Yaskawa INFORM job: R1_W39(90,0)R2.JBI

/JOB
//NAME R1_W39(90,0)R2
///FOLDERNAME KRIS-SCIANA
//POS
///NPOS 43,43,0,0,0,0
///TOOL 0
///POSTYPE PULSE
///PULSE
C00000=48919,5665,-78085,33957,84829,-60043
C00001=76192,72700,-3611,7580,89499,-58244
C00002=85002,90670,26729,6577,108191,-2594
C00003=82773,103392,47657,9044,108090,-2765
C00004=80348,95814,37890,14264,107528,-2580
C00005=80254,94172,37553,14217,106925,-2684
C00006=81389,106350,52541,15889,109549,-1922
C00007=88376,91776,33541,16145,112345,900
C00008=84647,97242,43547,26530,112715,1712
C00009=80535,96727,39662,19290,111179,-13264
C00010=80533,98698,38722,19533,112685,-13001
C00011=95804,88670,27983,-9101,104845,39456
C00012=93260,116784,65555,-9230,104296,50461
C00013=88788,88191,28703,620,100303,50675
C00014=93687,111856,59478,-9313,105536,50507
C00015=89184,93395,34979,471,102669,51670
C00016=95648,113896,64634,-12639,107588,50809
C00017=91118,114335,62249,-3400,106342,50920
C00018=94799,78029,20878,-7231,106457,51217
C00019=94179,105834,52955,-9270,106688,50794
C00020=97616,95145,42128,-15247,107009,50700
C00021=97568,79271,23775,-13354,106025,50913
C00022=97503,98351,37938,-14194,113675,56454
C00023=97503,100031,37397,-14345,114836,56304
C00024=130465,98764,47484,-38638,104472,-12047
C00025=128682,99899,51858,-38063,102058,-11895
C00026=125592,100494,53893,-37558,100021,-12435
C00027=117769,53841,-3568,-7004,89352,-33862
C00028=118319,55966,-2495,-7211,89822,-33727
C00029=127393,85542,37674,-37833,96354,-10529
C00030=118983,88052,33036,-15664,100505,-10201
C00031=114637,82539,25445,-1803,99860,-9026
C00032=114316,82458,25346,-216,99794,-11375
C00033=114685,80246,17709,-453,103292,-11364
C00034=111320,72755,14674,9080,100113,-13386
C00035=111645,74192,16353,7527,99507,-12765
C00036=112489,77538,20103,4175,98402,-12017
C00037=114786,72045,10431,-220,101192,-12172
C00038=116347,75543,8692,-605,104066,-11721
C00039=119316,88943,15862,706,106612,-10309
C00040=69963,28472,-55800,11354,82569,-11117
C00041=61683,17043,-76984,-12013,99317,-2721
C00042=8337,141,-97195,-54,99052,-6651
BC00000=111331,480623,1075175
BC00001=111331,480623,1075175
BC00002=156339,486365,1075175
BC00003=156270,481563,1075172
BC00004=156256,480588,1075175
BC00005=156256,480588,1075175
BC00006=156270,481563,1075172
BC00007=156270,481563,1075172
BC00008=156270,481563,1075172
BC00009=133619,478240,1075175
BC00010=135738,482219,1075175
BC00011=156256,480588,1075175
BC00012=156256,480588,1075171
BC00013=156256,480588,1075169
BC00014=156256,480588,1075171
BC00015=156256,480588,1075169
BC00016=156256,480588,1075169
BC00017=156256,480588,1075169
BC00018=156256,480589,1075170
BC00019=156256,480588,1075169
BC00020=156256,480589,1075168
BC00021=156256,480590,1075168
BC00022=156256,480588,1075171
BC00023=156256,480588,1075171
BC00024=264781,512151,1075175
BC00025=264781,512151,1075175
BC00026=264781,512151,1075175
BC00027=264644,511631,1075175
BC00028=264644,511631,1075175
BC00029=264781,512151,1075175
BC00030=264781,512151,1075175
BC00031=264781,512151,1075175
BC00032=264781,512151,1075175
BC00033=264781,512151,1075175
BC00034=264782,512151,1075173
BC00035=264782,512151,1075172
BC00036=264782,512151,1075173
BC00037=264782,512151,1075173
BC00038=264782,512151,1075173
BC00039=264782,512151,1075173
BC00040=86452,480608,1075173
BC00041=130207,480608,1075173
BC00042=130207,555252,1075173
//INST
///DATE 2024/03/27 17:42
///ATTR SC,RW
///GROUP1 RB1,BS1
NOP
'r2_W39(90,0)
'Path S818
MOVJ C00000 BC00000 VJ=30.00
MOVJ C00001 BC00001 VJ=50.00
SFTOF
MOVJ C00002 BC00002 VJ=30.00
MOVL C00003 BC00003 V=100.0 PL=0
REFP 1 C00004 BC00004
REFP 2 C00005 BC00005
MACRO1 MJ#(0) ARGF7
ARCON
MOVL C00006 BC00006 V=10.0
MOVL C00007 BC00007 V=10.0
MOVL C00008 BC00008 V=10.0
ARCOF
MOVL C00009 BC00009 V=100.0
MOVL C00010 BC00010 V=100.0
SFTOF
'COMMENT
MOVL C00011 BC00011 V=100.0
COMM MOVL C00012 BC00012 V=100.0 PL=0  //OLD POSITION
MOVL C00013 BC00013 V=100.0 PL=0
MACRO1 MJ#(0) ARGF7
ARCON
COMM MOVL C00014 BC00014 V=10.0  //OLD POSITION
MOVL C00015 BC00015 V=10.0
COMM MOVL C00016 BC00016 V=10.0
MOVL C00017 BC00017 V=10.0
COMM MOVL C00018 BC00018 V=10.0  //OLD POSITION
MOVL C00019 BC00019 V=10.0
ARCON
MOVL C00020 BC00020 V=10.0
MOVL C00021 BC00021 V=10.0
ARCOF
SFTOF
MOVL C00022 BC00022 V=100.0
'W53
SFTOF
MOVJ C00023 BC00023 VJ=20.00
MOVJ C00024 BC00024 VJ=20.00
MOVL C00025 BC00025 V=83.3
MOVL C00026 BC00026 V=50.0
REFP 1 C00027 BC00027
REFP 2 C00028 BC00028
MACRO1 MJ#(0) ARGF7
ARCON
MOVL C00029 BC00029 V=8.3
MOVL C00030 BC00030 V=8.3
MOVL C00031 BC00031 V=8.3
MOVL C00032 BC00032 V=8.3
ARCOF
MOVL C00033 BC00033 V=83.3
MOVL C00034 BC00034 V=83.3
ARCON
MOVL C00035 BC00035 V=8.3
MOVL C00036 BC00036 V=8.3
ARCOF
MOVL C00037 BC00037 V=250.0
MOVJ C00038 BC00038 VJ=100.00
MOVJ C00039 BC00039 VJ=100.00
MOVJ C00040 BC00040 VJ=80.00
MOVJ C00041 BC00041 VJ=100.00
MOVJ C00042 BC00042 VJ=100.00
SFTOF
END
